TYPE ST_VTUG :
STRUCT
	sol_A: BOOL;
	sol_B: BOOL;
END_STRUCT
END_TYPE

(* stored: Version 1.1.0.1, ProductVersion 3.1.4024.12
   DUT ST_VTUG: Id {b828fe01-4566-44dc-852a-62a2f9043997} *)
